{attribute 'GeneratedUsingTerminal: AT2026-0250-0020'}
{attribute addProperty BoxType "AT2026-0250-0020"}
{attribute addProperty Id "A_0078_AT2001_5250_0019_AT2001_5250AT2001_33A3DF1B80"}
{attribute addProperty CRC "2918768554"}
{attribute addProperty Size "80"}
TYPE A_0066_AT2026_0250_0020_AT2026_0250_ADF8DFAA EXTENDS AT2026_2EA6C9BF :
STRUCT
	{attribute addProperty Name "A_0078_AT2001_5250_0019_AT2001_5250"}
	{attribute addProperty PreviousPort "A_0066(AT2026-0250-0020) (AT2026-0250) : B"}
	A_0078_AT2001_5250_0019_AT2001_5250 : AT2001_33A3DF1B;
END_STRUCT
END_TYPE

(* stored: Version 1.2.0.0, ProductVersion 3.1.4024.9
   DUT A_0066_AT2026_0250_0020_AT2026_0250_ADF8DFAA: Id {0b77e71d-854e-4388-991b-41a8e39ce2fb} *)
